FUNCTION AscendingBubbleSort : BOOL
VAR_INPUT
END_VAR
VAR
	i: DINT;
	j: DINT;
	swap: INT;
	Swapped: BOOL;
END_VAR
VAR_IN_OUT
	ArrayToSort : array[*] of int;
END_VAR

FOR i := 0 TO UPPER_BOUND(ArrayToSort,1) DO
	Swapped := FALSE;
	FOR j := 0 TO (UPPER_BOUND(ArrayToSort,1) -1) DO
		IF ArrayToSort[j] > ArrayToSort[j+1] THEN
			swap := ArrayToSort[j];
			ArrayToSort[j] := ArrayToSort[j + 1];
			ArrayToSort[j+1] := swap;
			Swapped := TRUE;
		END_IF
	END_FOR
	IF NOT Swapped THEN
		EXIT;
	END_IF
END_FOR

END_FUNCTION

(* stored: Version 1.1.0.1, ProductVersion 3.1.4024.12
   POU AscendingBubbleSort: Id {829529fb-9434-48fd-95a9-152a1b6d6103}, SpecialFunc None *)
